// TIA Portal V21 export
VAR_GLOBAL   // PLC tag table "K_Pid"
END_VAR
VAR_GLOBAL CONSTANT   // user constants
   K_Pid_RaffreddamentoAcqua : Int := 1;
   K_Pid_RiscaldamentoAcqua : Int := 2;
   K_Pid_PompaMono : Int := 3;
   K_Pid_PompaPistoni : Int := 4;
   K_Pid_RiscaldamentoProdotto : Int := 5;
END_VAR
